INTERFACE IMover

PROPERTY AxisRef : reference to axis_ref
GET
END_GET
END_PROPERTY

METHOD DisableAxis : BOOL
VAR_INPUT
END_VAR
END_METHOD

METHOD EnableAxis : BOOL
VAR_INPUT
END_VAR
END_METHOD

METHOD HaltAxis : BOOL
VAR_INPUT
END_VAR
END_METHOD

PROPERTY IdentInGroup : int
GET
END_GET
SET
END_SET
END_PROPERTY

METHOD isAtPosition : BOOL
VAR_INPUT
	position : MC_LREAL;
END_VAR
END_METHOD

METHOD isDetected : BOOL
VAR_INPUT
END_VAR
END_METHOD

METHOD isEnabled : BOOL
VAR_INPUT
END_VAR
END_METHOD

METHOD MoveTo : BOOL
VAR_INPUT
	Position : MC_LREAL;
	Velocity : MC_LREAL;
	BackwardMove : BOOL;
END_VAR
END_METHOD

METHOD ResetAxis : BOOL
VAR_INPUT
END_VAR
END_METHOD

END_INTERFACE

(* stored: Version 1.1.0.1, ProductVersion 3.1.4024.6
   Itf IMover: Id {0e30beea-f524-44e1-ae12-0e02166014dd}
   Property AxisRef: Id {32f17bdd-a939-4d9e-98cc-91a8a53a6910}
   Get Get: Id {69e35166-9a24-48e6-815a-1166e16ded53}
   Method DisableAxis: Id {689f2355-5608-4781-bf9f-baf702db6fd8}
   Method EnableAxis: Id {e787a67b-7883-495a-9a3a-341e1daf5c57}
   Method HaltAxis: Id {ebcb5f64-4a36-49eb-91f7-3a5c2f6ad022}
   Property IdentInGroup: Id {3957605a-f901-42a3-a167-84d75e8b2803}
   Get Get: Id {0cec0afa-43ba-4ae0-9403-f6ae41b75c8f}
   Set Set: Id {1acbbc53-227d-4433-984f-d50b20a1b1d3}
   Method isAtPosition: Id {94cda122-57e0-415e-a76d-4df809bff294}
   Method isDetected: Id {5b28002b-408a-49b8-8a2d-6fa82833fceb}
   Method isEnabled: Id {aedc5d49-1b43-4d77-a9fc-9b26bd3b8a96}
   Method MoveTo: Id {ad2ef999-10e1-4863-90d6-0a9a5ca633ef}
   Method ResetAxis: Id {73269db4-aebb-4b1b-91e1-629b242c142c} *)
